TEXTLIST ParameterTextList
  1 = 'CommandedPosition'
  2 = 'SWLimitForward'
  3 = 'SWLimitBackward'
  4 = 'EnableLimitForward'
  5 = 'EnableLimitBackward'
  6 = 'EnablePositionLagMonitoring'
  7 = 'MaxPositionLag'
  8 = 'AxisMaxVelocity'
  10 = 'ActualVelocity'
  11 = 'CommandedVelocity'
  12 = 'AxisDefaultAcceleration'
  14 = 'AxisDefaultDeceleration'
  16 = 'AxisDefaultJerk'
  1000 = 'AxisId'
  1001 = 'AxisManualVelocitySlow'
  1002 = 'AxisManualVelocityFast'
  1009 = 'AxisRapidTraverseVelocity'
  1012 = 'AxisVelocityToCam'
  1013 = 'AxisVelocityFromCam'
  1014 = 'AxisJogIncrementForward'
  1015 = 'AxisJogIncrementBackward'
  1022 = 'MaxPositionLagFilterTime'
  1023 = 'AxisEnPositionRangeMonitoring'
  1024 = 'AxisPositionRangeWindow'
  1025 = 'AxisEnTargetPositionMonitoring'
  1026 = 'AxisTargetPositionWindow'
  1027 = 'AxisTargetPositionMonitoringTime'
  1028 = 'AxisEnInTargetTimeout'
  1029 = 'AxisInTargetTimeout'
  1030 = 'AxisEnMotionMonitoring'
  1031 = 'AxisMotionMonitoringWindow'
  1032 = 'AxisMotionMonitoringTime'
  1033 = 'AxisDelayTimeVeloPosition'
  1034 = 'AxisEnLoopingDistance'
  1035 = 'AxisLoopingDistance'
  1038 = 'AxisEnDataPersistence'
  1039 = 'AxisRefVeloOnRefOutput'
  1040 = 'AxisOverrideType'
  1042 = 'AxisEncoderOffset'
  1043 = 'AxisEncoderDirectionInverse'
  1044 = 'AxisEncoderMask'
  1045 = 'AxisEncoderModuloValue'
  1046 = 'AxisModuloToleranceWindow'
  1047 = 'AxisEnablePosCorrection'
  1048 = 'AxisPosCorrectionFilterTime'
  1049 = 'AxisUnitInterpretation'
  1050 = 'AxisMotorDirectionInverse'
  1051 = 'AxisCycleTime'
  1052 = 'AxisFastStopSignalType'
  1053 = 'AxisFastAcc'
  1054 = 'AxisFastDec'
  1055 = 'AxisFastJerk'
  1056 = 'AxisEncoderScalingNumerator'
  1057 = 'AxisEncoderScalingDenominator'
  1058 = 'AxisMaximumAcceleration'
  1059 = 'AxisMaximumDeceleration'
  1060 = 'AxisVeloJumpFactor'
  1061 = 'AxisToleranceBallAuxAxis'
  1062 = 'AxisMaxPositionDeviationAuxAxis'
  1063 = 'AxisErrorPropagationMode'
  1064 = 'AxisErrorPropagationDelay'
  1065 = 'AxisCoupleSlaveToActualValues'
  1066 = 'AxisAllowMotionCmdToSlaveAxis'
  1067 = 'AxisAllowMotionCmdToExtSetAxis'
  1068 = 'AxisEncoderSubMask'
  1069 = 'AxisEncoderReferenceSystem'
  1070 = 'AxisEncoderPositionFilterPT1'
  1071 = 'AxisEncoderVelocityFilterPT1'
  1072 = 'AxisEncoderAccelerationFilterPT1'
  1073 = 'AxisEncoderMode'
  1074 = 'AxisEncoderHomingInvDirCamSearch'
  1075 = 'AxisEncoderHomingInvDirSyncSearch'
  1076 = 'AxisEncoderHomingCalibValue'
  1077 = 'AxisEncoderReferenceMode'
  1078 = 'AxisRefVeloOutputRatio'
  1079 = 'AxisDrivePositionOutputScaling'
  1080 = 'AxisDriveVelocityOutputScaling'
  1081 = 'AxisDriveVelocityOutputDelay'
  1082 = 'AxisDriveMinOutputLimitation'
  1083 = 'AxisDriveMaxOutputLimitation'
  1084 = 'AxisTorqueInputScaling'
  1085 = 'AxisTorqueInputFilterPT1'
  1086 = 'AxisTorqueDerivationInputFilterPT1'
  1087 = 'AxisTorqueOutputScaling'
  1088 = 'AxisTorqueOutputDelay'
  1089 = 'AxisAccelerationOutputScaling'
  1090 = 'AxisAccelerationOutputDelay'
  1091 = 'AxisDrivePositionOutputSmoothFilterType'
  1092 = 'AxisDrivePositionOutputSmoothFilterTime'
  1093 = 'AxisDrivePositionOutputSmoothFilterOrder'
  1094 = 'AxisDriveMode'
  1095 = 'AxisDriftCompensationOffset'
  1096 = 'AxisPositionControlKv'
  1097 = 'AxisCtrlVelocityPreCtrlWeight'
  1098 = 'AxisControllerMode'
  1099 = 'AxisCtrlAutoOffset'
  1100 = 'AxisCtrlAutoOffsetTimer'
  1101 = 'AxisCtrlAutoOffsetLimit'
  1102 = 'AxisSlaveCouplingControlKcp'
  1103 = 'AxisCtrlOutputLimit'
  2000 = 'AxisTargetPosition'
  2001 = 'AxisRemainingTimeToGo'
  2002 = 'AxisRemainingDistanceToGo'
  3000 = 'AxisGearRatio'
  4000 = 'NcSafCycleTime'
  4001 = 'NcSvbCycleTime'
   = ''
END_TEXTLIST

(* stored: Version 1.1.0.1, ProductVersion 3.1.4024.11
   TextList ParameterTextList: Id {89b0f5ae-06d0-4e0b-a194-a2a3afdf3247} *)
